Universal Robots PolyScope program: preprod_v3.urp

Program preprod_v3 (installation=preprod directory=/home/ur/ursim-current/programs/programs.UR10/Preproduction createdIn=3.14.1.1031110 lastSavedIn=3.14.1.1031110 robotSerialNumber=2018309999)
Calibrated DH parameters: a=[-0.000013, -0.603836, -0.568298, -0.000064, 0.000091, 0]; d=[0.128008, 14.734433, -5.969991, -8.600746, 0.115672, 0.092215]; alpha=[1.570325, -0.007027, -0.006659, 1.569356, -1.5695, 0]; deltaTheta=[-0.000047, -0.169823, 0.067411, 0.102409, -0.00005, 0.00003]
InitVariablesNode variables(variable(name=last_task, expression=0), variable(name=print1, expression=False), variable(name=print2, expression=False), variable(name=print3, expression=False), variable(name=print_enable, expression=False), variable(name=vision_pos, expression=p[0,0,0,0,0,0]))
BeforeStart
  Script file /programs/Preproduction/readme.script
    | # SETUP INFO
    | 
    | # 1. Configure TCP
    | # 2. Calibrate to vision plane
    | # 3. Set the home position
    | # 4. Set variables at setup
    | 
    | # stack_ry - corresponds to tool rotation vector relative to stack
    | # print_width - width of the print label
    | # printer_width - width of the printer head
    | # ramp_distance - how far to reach constant speed
    | # clearance - how far away are we printing from the stack
    | # box_to_PA_XY - box coord to print area
    | # stack_a_to_ref - adjusts the vision plane calibration discrepancies
    | # TE_L2R - Task enum left to right
  Folder Config
    'Printing Properties'
    clearance := 0.04
    ramp_dist := 0.1
    trigger_range := 0.003
    L2R_trig_dist := 0.01
    R2L_trig_dist := 0.058
    'The tcp rotation components relative to stack'
    stack_rx := 0
    stack_ry := -d2r(180)
    stack_rz := 0
    'Reference Frame Tuning'
    box_to_pa_XY := p[0,0,0,0,0,0]
    stack_a_to_ref := p[0,0,0,0,0,0]
    stack_b_to_ref := p[0,0,0,0,0,0]
  Folder Config Static
    'Physical Properties'
    print_width := 0.04
    printer_width := 0.125
    'Task Enumeration'
    TE_L2R := 1
    TE_R2L := 2
  Folder Config Calcs
    pa_x_clear := (print_width+printer_width)/2
    runover := pa_x_clear+ramp_dist
  Folder Restart Checks
    tasks_equal := task≟current_task
    tasks_printing := task≠0 and current_task≠0 print_enable
    restart_task := GP_bool_in[64] and ( not tasks_equal) and tasks_printing
    resume_task := start_continue and tasks_equal and tasks_printing
    print_enable := False
  Folder Keep current pos as home
    sp := get_actual_joint_positions()
    MoveJ speed 60 deg/s, acceleration 80 deg/s^2 (useActiveTCP=true)
      Waypoint Waypoint (Variable): variable=sp
  Folder Reset bits
    Set DigitalOutput pin=task_done; digitalValue=0
    Set DigitalOutput pin=task_active; digitalValue=0
    Set ExpressionOutput pin=current_task; expression=0
    Set DigitalOutput pin=moving_home; digitalValue=0
    Set DigitalOutput pin=homed; digitalValue=0
Robot Program (runOnlyOnce=false)
  If gantry_in_pos_a or GP_bool_in[75]
    If cancel_home
      Call PreTask
      Call MoveHome
    ElseIf task≟TE_L2R or task≟TE_R2L
      Call PreTask
      Call StartTask
      Call SetWaypoints
      Call SanitiseInputs
      Call MoveWaypoints
      Call FinishTask
SubProgram -> PreTask
SubProgram -> MoveHome
SubProgram -> StartTask
SubProgram -> SetWaypoints
SubProgram -> SanitiseInputs
SubProgram -> MoveWaypoints
SubProgram -> FinishTask
Thread Thread_1 (runOnlyOnce=false)
  'Monitors X position for printing'
  If print_enable
    vision_pos := pose_trans(pose_inv(reference), get_actual_tcp_pose())
    print1 := norm(vision_pos[0] - (PA1[0]-xm*(trigger_offset-trigger_range/2))) ≤ trigger_range
    print2 := norm(vision_pos[0] - (PA2[0]-xm*(trigger_offset-trigger_range/2))) ≤ trigger_range
    print3 := norm(vision_pos[0] - (PA3[0]-xm*(trigger_offset-trigger_range/2))) ≤ trigger_range
    If print1 or print2 or print3
      Set SingleDigitalPulseActionState SingleDigitalPulseActionState(hiPulseInSeconds=0.05, pin=GP_bool_out[68])
      Set SingleDigitalPulseActionState SingleDigitalPulseActionState(hiPulseInSeconds=0.05, pin=config_out[0])
  Script: sync()
SubProgram PreTask (keepSynchronizedWithDisk=false)
  If not (GP_bool_in[74] xor GP_bool_in[75])
    Popup Warning (haltProgram=false message=Err: Gantry not in pos inputType=Text)
    Halt
  ElseIf GP_bool_in[74]
    reference := pose_add(stack_b, stack_b_to_ref)
  ElseIf GP_bool_in[75]
    reference := pose_add(stack_a, stack_a_to_ref)
  'Where is the miminimum Z relative to current pos'
  vision_pos_ex := pose_trans(pose_inv(reference), get_actual_tcp_pose())
  vision_pos_ex := pose_add(vision_pos_ex, p[0, 0, 2*clearance + GP_float_in[9] - vision_pos_ex[2], 0, 0, 0])
  CLEAR := pose_trans(reference, vision_pos_ex)
SubProgram MoveHome (keepSynchronizedWithDisk=false)
  Set ExpressionOutput pin=current_task; expression=0
  Set DigitalOutput pin=task_done; digitalValue=0
  Set DigitalOutput pin=task_active; digitalValue=0
  If not homed
    Set ExpressionOutput pin=moving_home; expression=True
    MoveL speed 500 mm/s, acceleration 500 mm/s^2 (useActiveTCP=true) feature=Base
      Waypoint home: TCP in base x=-341.446 y=-425.238 z=1068.774 mm, rx=-0.7092 ry=-1.7644 rz=1.7532 rad; joints [-4.235, -118.304, 92.312, -154.015, -40.459, -0.894] deg; flange x=-300.566 y=-212.476 z=1032.647 mm, rx=-0.7092 ry=-1.7644 rz=1.7532 rad
        Until REACHED_WAYPOINT (allowActions=true)
          Set DigitalOutput pin=homed; digitalValue=1
    Set ExpressionOutput pin=moving_home; expression=False
SubProgram StartTask (keepSynchronizedWithDisk=false)
  Set ExpressionOutput pin=current_task; expression=GP_int_in[0]
  Set DigitalOutput pin=task_active; digitalValue=1
SubProgram SetWaypoints (keepSynchronizedWithDisk=false)
  Folder Set Ordering
    B2 := p[GP_float_in[1], GP_float_in[3], GP_float_in[6], 0, 0, 0]
    If current_task≟TE_L2R
      'Left to right (+ive)'
      xm := 1
      B1 := p[X1, Y, Z, 0, 0, 0]
      B3 := p[X3, Y, Z, 0, 0, 0]
      trigger_offset := pa_x_clear+L2R_trig_dist
    ElseIf current_task≟TE_R2L
      'Right to left (-ive)'
      xm := -1
      B1 := p[X3, Y, Z, 0, 0, 0]
      B3 := p[X1, Y, Z, 0, 0, 0]
      trigger_offset := pa_x_clear+R2L_trig_dist
  Folder Print Area Vars
    'Move the print areas relative to given box'
    PA1 := pose_add(B1, box_to_pa_XY)
    PA2 := pose_add(B2, box_to_pa_XY)
    PA3 := pose_add(B3, box_to_pa_XY)
  Folder Calculate Waypoints
    'xm represents with flow, -xm represents against flow'
    PA1_EN := pose_add(PA1, p[-runover*xm, 0, clearance, stack_rx, stack_ry, stack_rz])
    PA3_EX := pose_add(PA3, p[+runover*xm, 0, clearance, stack_rx, stack_ry, stack_rz])
    'Rotation?'
    APPROACH := pose_add(PA1_EN, p[0, 0, 2*clearance + GP_float_in[9] - PA1_EN[2], 0, 0, 0])
  Folder Reference Base
    PA1_EN := pose_trans(reference, PA1_EN)
    PA3_EX := pose_trans(reference, PA3_EX)
    APPROACH := pose_trans(reference, APPROACH)
SubProgram SanitiseInputs (keepSynchronizedWithDisk=false)
  ''
SubProgram MoveWaypoints (keepSynchronizedWithDisk=false)
  'Position before the move'
  If homed
    MoveL speed 500 mm/s, acceleration 2000 mm/s^2 (useActiveTCP=true) feature=Base
      Set ExpressionOutput pin=homed; expression=False
      Waypoint Waypoint (Variable): motionParameters(blendRadius=0.04); variable=APPROACH
        Until EXPRESSION (allowActions=false) ExpressionBranch=GP_bool_in[76]
      Waypoint Waypoint (Variable): motionParameters(blendRadius=0.05); variable=PA1_EN
        Until EXPRESSION (allowActions=false) ExpressionBranch=GP_bool_in[76]
  ElseIf resume_task
    'Resume from current position'
    Set ExpressionOutput pin=homed; expression=False
  ElseIf last_task≟TE_L2R and current_task≟TE_R2L and  not restart_task
    'L2R -> R2L'
    Set ExpressionOutput pin=homed; expression=False
    MoveL speed 500 mm/s, acceleration 2000 mm/s^2 (useActiveTCP=true) feature=Base
      Waypoint Waypoint (Variable): motionParameters(blendRadius=0.05); variable=PA1_EN
        Until EXPRESSION (allowActions=false) ExpressionBranch=GP_bool_in[76]
  Else 
    MoveL speed 500 mm/s, acceleration 2000 mm/s^2 (useActiveTCP=true) feature=Base
      Set ExpressionOutput pin=homed; expression=False
      Waypoint Waypoint (Variable): motionParameters(blendRadius=0.04); variable=CLEAR
        Until EXPRESSION (allowActions=false) ExpressionBranch=GP_bool_in[76]
      Waypoint Waypoint (Variable): motionParameters(blendRadius=0.04); variable=APPROACH
        Until EXPRESSION (allowActions=false) ExpressionBranch=GP_bool_in[76]
      Waypoint Waypoint (Variable): motionParameters(blendRadius=0.05); variable=PA1_EN
        Until EXPRESSION (allowActions=false) ExpressionBranch=GP_bool_in[76]
  'Move Across'
  MoveL speed 500 mm/s, acceleration 3000 mm/s^2 (useActiveTCP=true) feature=Base
    print_enable := True
    Waypoint Waypoint (Variable): variable=PA3_EX
      Until EXPRESSION (allowActions=false) ExpressionBranch=GP_bool_in[76]
    print_enable := False
  resume_task := False
SubProgram FinishTask (keepSynchronizedWithDisk=false)
  'Acknowledgement sequence with PLC'
  last_task := current_task
  Set DigitalOutput pin=task_active; digitalValue=0
  Set DigitalOutput pin=task_done; digitalValue=1
  Wait Condition expression=task≟0 or cancel_home
  Set ExpressionOutput pin=current_task; expression=0
  Set DigitalOutput pin=task_done; digitalValue=0
